Staubli VAL3: getTime.pgx

public program getTime(num& x_nTime[], bool x_bCycle, num x_nIndex)
begin
  // get the time DATA
  if x_bCycle
    // get the time DATA
    x_nTime=pt:tTraj[sItemCycle].tData[x_nIndex].tSuper.nTime
  else
    // get the time DATA
    x_nTime=pEditPoint.tData[x_nIndex].tSuper.nTime
  endIf
end
